FUNCTION_BLOCK FB_rotaButtonDetect
VAR_INPUT
END_VAR
VAR_OUTPUT
END_VAR
VAR
	m_rotaButtonUpOnCounts :INT :=0;
	m_rotaButtonUpOnCountThres :INT :=50;
	m_rotaButtonDownOnCounts :INT :=0;
	m_rotaButtonDownOnCountThres :INT :=-50;
END_VAR

// check if instrument is on
METHOD run : UDINT
VAR_INPUT
	IOValue :UDINT;
END_VAR
// 
IF 1=(IOValue AND 16#01) OR 2=(IOValue AND 16#02) THEN
	m_rotaButtonUpOnCounts :=MIN(m_rotaButtonUpOnCounts +1,m_rotaButtonUpOnCountThres);
ELSE
	m_rotaButtonUpOnCounts :=0;
END_IF

IF m_rotaButtonUpOnCounts >= m_rotaButtonUpOnCountThres THEN
	run := IOValue;
ELSE
	run := 0;
END_IF
END_METHOD

END_FUNCTION_BLOCK

(* stored: Version 1.1.0.1, ProductVersion 3.1.4024.11
   POU FB_rotaButtonDetect: Id {30693b56-bccc-471c-9eb1-da466ba07a53}, SpecialFunc None
   Method run: Id {c6d6ce7b-49be-4d76-8341-ace7fb023bb6} *)
